FUNCTION_BLOCK FB_AnalogOut0_10V
VAR_INPUT
	EngInput				: REAL;
	EngLowLimit				: REAL; (*Low limit*)
	EngUpperLimit 			: REAL; (*Upper limit*)
END_VAR
VAR_OUTPUT
END_VAR
VAR
	VOut 					: REAL;
	RawOut 					AT %Q* : INT;
END_VAR

VOut		:= 10/(EngUpperLimit-EngLowLimit)*(EngInput--EngLowLimit);
RawOut		:= REAL_TO_INT(32767.0/(EngUpperLimit-EngLowLimit)*(EngInput--EngLowLimit));

END_FUNCTION_BLOCK

(* stored: Version 1.1.0.1, ProductVersion 3.1.4020.12
   POU FB_AnalogOut0_10V: Id {3f2e3f66-2671-4139-8e47-c690c7bde4e3}, SpecialFunc None *)
